{attribute addProperty BoxType "AMP8000-0030-0103-0103"}
{attribute addProperty Id "FSOEAT %Q*FSOE_A616C3D6567"}
{attribute addProperty CRC "2044734574"}
{attribute addProperty SizeInBites "56"}
{attribute addProperty SizeInBytes "7"}
TYPE FSoE_Slave_Connection_1_Master_Message_79E02C6E :
STRUCT
	{attribute addProperty Name "FSOE"}
	FSOE AT %Q* : FSOE_A616C3D6;
END_STRUCT
END_TYPE

(* stored: Version 1.2.0.0, ProductVersion 3.1.4024.9
   DUT FSoE_Slave_Connection_1_Master_Message_79E02C6E: Id {0059aed6-dab4-435e-a4ac-eceee098cb80} *)
